(* IEC 61131-3 sources: AXOpen/src/integrations/ctrl/src/IntegrationTests, 1 file *)

(* ---- integrationtests.st ---- *)
NAMESPACE IntegrationTests
    CLASS PUBLIC Integrations
        VAR PUBLIC
             Probers : ProbersTestContext;
             DataExchangeLightTestsContext : IntegrationLightDirect.DataExchangeLightTestsContext;
             DataFragmentContext : IntegrationAxoDataFramentsExchange.AxoDataFragmentExchangeContext;
             DM : IntegrationLightDirect.DataManager;
        END_VAR

        METHOD PUBLIC Run
            Probers.Run();
            DM.Run(DataExchangeLightTestsContext);
            DataExchangeLightTestsContext.InjectDM(DM);
            DataExchangeLightTestsContext.Run();
            DataFragmentContext.Run();
        END_METHOD
    END_CLASS
END_NAMESPACE
